(* Logix 5000 project; controller TEC_81 vendor 1 type 14 code 148 rev 36.11; software revision 36.00; part 3 of 4 *)
(* tags used below, declared in another part *)
   Abrir_Prensa_CNC_2 : BOOL;   // START CYCLE CNC 2
   AbrirInterlock_conveyor_Control : BOOL;
   AbrirInterlock_conveyor_Safety : BOOL;
   AbrirInterlock_Principal_Control : BOOL;
   AbrirInterlock_Principal_Safety : BOOL;
   Axis_1 : AXIS_CIP_DRIVE;
   Axis_2 : AXIS_CIP_DRIVE;   // Almacen 2
   Close_Griper_Fanuc : BOOL;   // Señal de Griper Cerrado Robot Fanuc
   Cmd_Axis_2 : BOOL;
   Cmd_Robot_Conv_1 : BOOL;
   Cmd_Robot_Conv_2 : BOOL;
   Cmd_YPickSafe_Alm1 : BOOL;
   Cmd_YPlaceSafe_Alm1 : BOOL;
   Cmd_YSafePos_Alm1 : BOOL;
   Cmd_YtoYOff_Alm1 : BOOL;
   Cmd_YtoYPick_Alm1 : BOOL;
   Cmd_YtoYPlace_Alm1 : BOOL;
   Cmd_YtoYPlaceOffset_Alm1 : BOOL;
   Consumeded_Signals_Conveyor_1_TEC_81 : DINT;
   Conveyor_1_Tomar_Pieza : BOOL;   // Señal del Conveyor 1 para Tomar Pieza Iniciar Ciclo
   Conveyor_2_Tomar_Pieza : BOOL;   // Señal del Conveyor 2 para Tomar Pieza Iniciar Ciclo
   Destino_Fanuc_Wait : BOOL;
   EStops_OK : BOOL;
   EStops_OK_External : DINT;
   Fanuc_Confirma_Dejar_Pieza : BOOL;   // Confirmación del Robot Fanuc para dejar la pieza
   Fanuc_Confirma_Retraido : BOOL;   // Señal de Fanuc en posición segura en Mesa Kuka
   Fanuc_Confirma_Tomar_Pieza : BOOL;   // Señal de Fanuc en posición para Tomar pieza
   From_Robot : FromRobot_v02;
   From_Wh2 : DINT;
   FromStorage1 : DINT;
   Home_Sensor : BOOL;
   Input_Reset_Almacen_1 : BOOL;
   Input_Reset_almacen_2 : BOOL;
   Input_Reset_Principal : BOOL;
   Input_Reset_Salida_1 : BOOL;
   Int_Robot_2 : INT;
   Interlocks_Ok : BOOL;
   LigthCurtain_ok : BOOL;
   MC_1_EStop : DCI_STOP;
   MC_1_EStop_Status : BOOL;
   MC_1_Interlock : DCI_STOP;
   MC_1_Interlock_Status : BOOL;
   MC_1_LigthCurtain : DCI_STOP;
   MC_1_LigthCurtain_Status : BOOL;
   MC_2_EStop : DCI_STOP;
   MC_2_EStop_Status : BOOL;
   MC_2_Interlock : DCI_STOP;
   MC_2_Interlock_Status : BOOL;
   MC_2_LightCurtain_Status : BOOL;
   MC_2_LigthCurtain : DCI_STOP;
   MC_3_EStop : DCI_STOP;
   MC_3_EStop_Status : BOOL;
   MC_4_EStop : DCI_STOP;
   MC_4_EStop_Status : BOOL;
   MC_5_EStop : DCI_STOP;
   MC_5_EStop_Status : BOOL;
   ok : BOOL;
   Open_Griper_Fanuc : BOOL;   // Señal De Griper Abierto Robot Fanuc
   Produced_Signals_TEC_81_Conveyor_1 : DINT;
   Puerta_Abierta_CNC_1 : BOOL;   // Sensor de Puerta Abierta en CNC 1 Conveyor 1
   Puerta_Abierta_CNC_2 : BOOL;   // Sensor de Puerta Abierta en CNC 2 Conveyor 2
   Reset_Almacen_1 : BOOL;
   Reset_almacen_2 : BOOL;
   Reset_Principal : BOOL;
   Reset_Salida_1 : BOOL;
   Retorno_Pieza_A_Conveyor_1 : BOOL;
   Robot_Step : DINT;
   Safety_FromTEC81 : Safety;
   SafetyReset_almacen_1 : BOOL;
   SafetyReset_almacen_2 : BOOL;
   SafetyReset_Principal : BOOL;
   SafetyReset_Salida_1 : BOOL;
   Sensor_Griper_Fanuc_Abierto : BOOL;   // Sensor Indicador Griper en Robot Fanuc Abierto
   Sensor_Griper_Fanuc_Cerrado : BOOL;   // Sensor Indicador Griper en Robot Fanuc Cerrado
   Sensor_Piston_2_Ext_Mesa : BOOL;   // Sensor de Pistón Extendido Centro de la Mesa Central
   Sensor_Piston_2_Ret_Mesa : BOOL;   // Sensor de Pistón Retraido Centro de la Mesa Central
   Signal_Fanuc_Tomar_Pieza_Conv_1 : BOOL;   // Señal para Tomar pieza desde el Conveyor 1 Hacia CNC
   Storage_1_Y_ActualPosition : REAL;
   Storage_2_Y_ActualPosition : REAL;
   Tec81_to_Wh2 : DINT;
   test_com : BOOL;   // bit e comunicacion
   TEst_Leaa_Sfty : DINT;
   To_Robot : ToRobot;
   TT : BOOL;

PROGRAM MainProgram   (* main routine MainRoutine *)

ROUTINE _01_Inputs   (* ladder *)
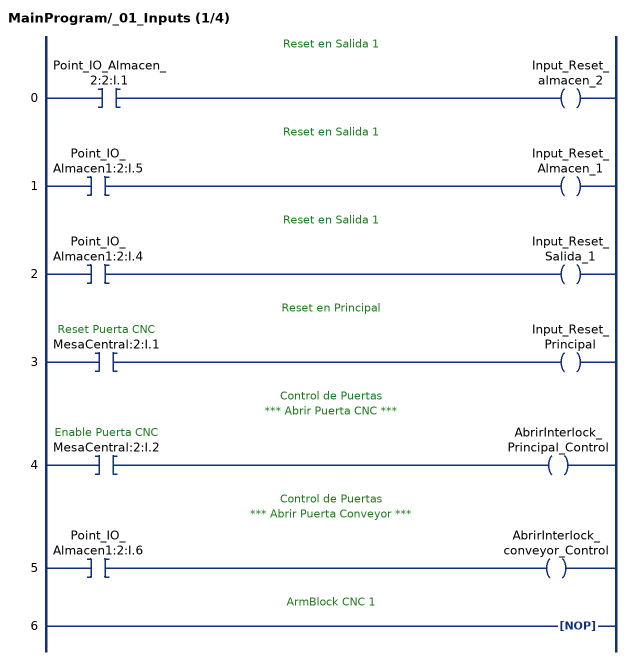
   // Reset en Salida 1
   0: XIC(Point_IO_Almacen_2:2:I.1)OTE(Input_Reset_almacen_2);
   // Reset en Salida 1
   1: XIC(Point_IO_Almacen1:2:I.5)OTE(Input_Reset_Almacen_1);
   // Reset en Salida 1
   2: XIC(Point_IO_Almacen1:2:I.4)OTE(Input_Reset_Salida_1);
   // Reset en Principal
   3: XIC(MesaCentral:2:I.1)OTE(Input_Reset_Principal);
   // Control de Puertas
   // *** Abrir Puerta CNC ***
   4: XIC(MesaCentral:2:I.2)OTE(AbrirInterlock_Principal_Control);
   // Control de Puertas
   // *** Abrir Puerta Conveyor ***
   5: XIC(Point_IO_Almacen1:2:I.6)OTE(AbrirInterlock_conveyor_Control);
   // ArmBlock CNC 1
   6: NOP();
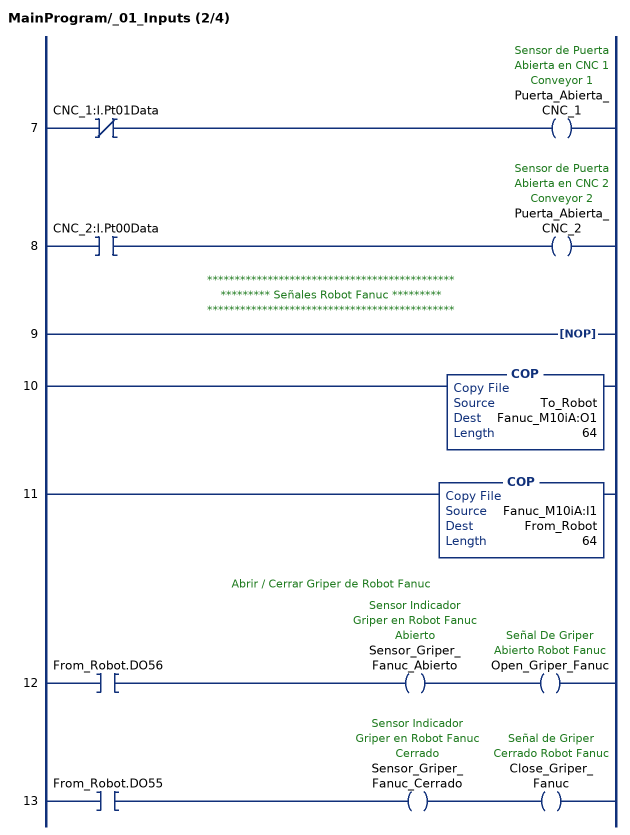
   7: XIO(CNC_1:I.Pt01Data)OTE(Puerta_Abierta_CNC_1);
   8: XIC(CNC_2:I.Pt00Data)OTE(Puerta_Abierta_CNC_2);
   // *********************************************
   // ********* Señales Robot Fanuc *********
   // *********************************************
   9: NOP();
   10: COP(To_Robot,Fanuc_M10iA:O1,64);
   11: COP(Fanuc_M10iA:I1,From_Robot,64);
   // Abrir / Cerrar Griper de Robot Fanuc
   12: XIC(From_Robot.DO56)OTE(Sensor_Griper_Fanuc_Abierto)OTE(Open_Griper_Fanuc);
   13: XIC(From_Robot.DO55)OTE(Sensor_Griper_Fanuc_Cerrado)OTE(Close_Griper_Fanuc);
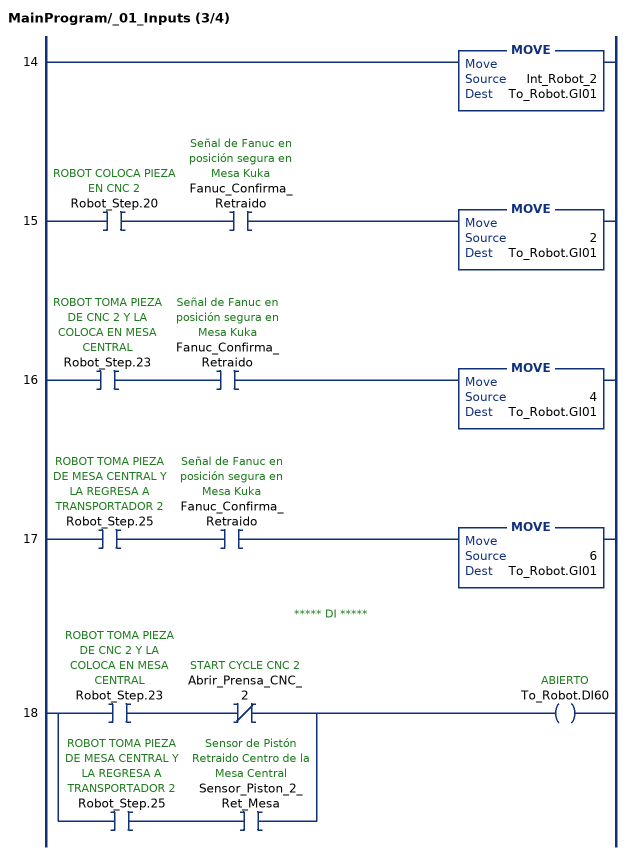
   14: MOVE(Int_Robot_2,To_Robot.GI01);
   15: XIC(Robot_Step.20)XIC(Fanuc_Confirma_Retraido)MOVE(2,To_Robot.GI01);
   16: XIC(Robot_Step.23)XIC(Fanuc_Confirma_Retraido)MOVE(4,To_Robot.GI01);
   17: XIC(Robot_Step.25)XIC(Fanuc_Confirma_Retraido)MOVE(6,To_Robot.GI01);
   // ***** DI *****
   18: [XIC(Robot_Step.23) XIO(Abrir_Prensa_CNC_2) ,XIC(Robot_Step.25) XIC(Sensor_Piston_2_Ret_Mesa) ]OTE(To_Robot.DI60);
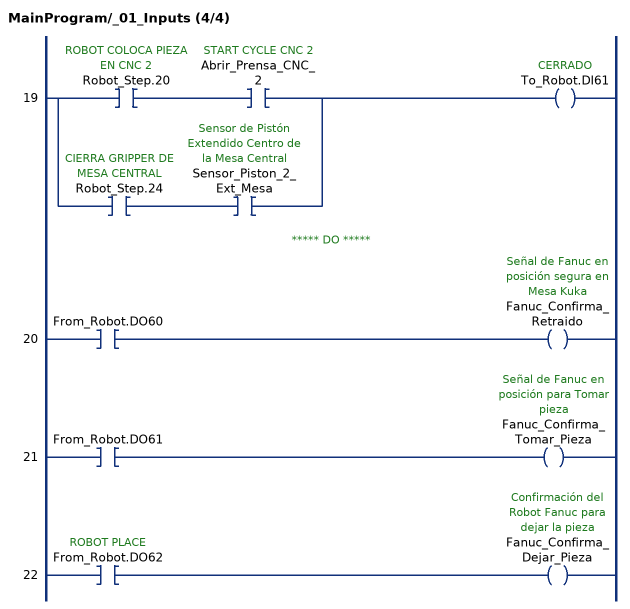
   19: [XIC(Robot_Step.20) XIC(Abrir_Prensa_CNC_2) ,XIC(Robot_Step.24) XIC(Sensor_Piston_2_Ext_Mesa) ]OTE(To_Robot.DI61);
   // ***** DO *****
   20: XIC(From_Robot.DO60)OTE(Fanuc_Confirma_Retraido);
   21: XIC(From_Robot.DO61)OTE(Fanuc_Confirma_Tomar_Pieza);
   22: XIC(From_Robot.DO62)OTE(Fanuc_Confirma_Dejar_Pieza);
END_ROUTINE

ROUTINE _06_Fanuc_States   (* ladder *)
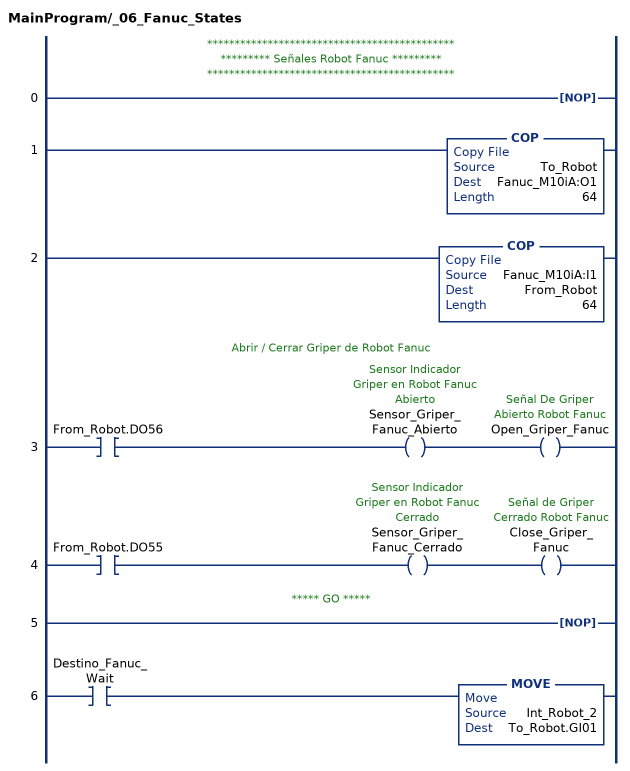
   // *********************************************
   // ********* Señales Robot Fanuc *********
   // *********************************************
   0: NOP();
   1: COP(To_Robot,Fanuc_M10iA:O1,64);
   2: COP(Fanuc_M10iA:I1,From_Robot,64);
   // Abrir / Cerrar Griper de Robot Fanuc
   3: XIC(From_Robot.DO56)OTE(Sensor_Griper_Fanuc_Abierto)OTE(Open_Griper_Fanuc);
   4: XIC(From_Robot.DO55)OTE(Sensor_Griper_Fanuc_Cerrado)OTE(Close_Griper_Fanuc);
   // ***** GO *****
   5: NOP();
   6: XIC(Destino_Fanuc_Wait)MOVE(Int_Robot_2,To_Robot.GI01);
END_ROUTINE

ROUTINE _08_Outputs   (* ladder *)
END_ROUTINE

ROUTINE _09_Resets   (* ladder *)
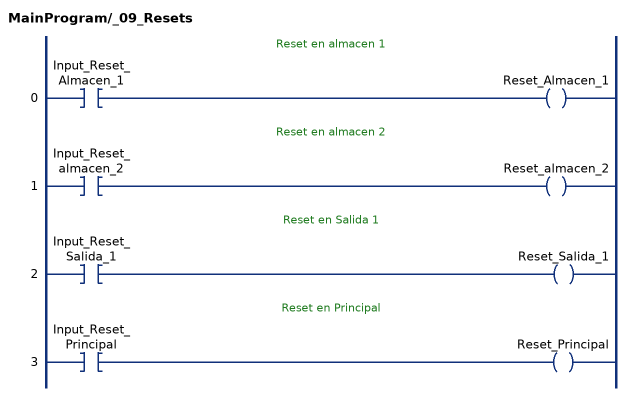
   // Reset en almacen 1
   0: XIC(Input_Reset_Almacen_1)OTE(Reset_Almacen_1);
   // Reset en almacen 2
   1: XIC(Input_Reset_almacen_2)OTE(Reset_almacen_2);
   // Reset en Salida 1
   2: XIC(Input_Reset_Salida_1)OTE(Reset_Salida_1);
   // Reset en Principal
   3: XIC(Input_Reset_Principal)OTE(Reset_Principal);
END_ROUTINE

ROUTINE _10_ExternalComm   (* ladder *)
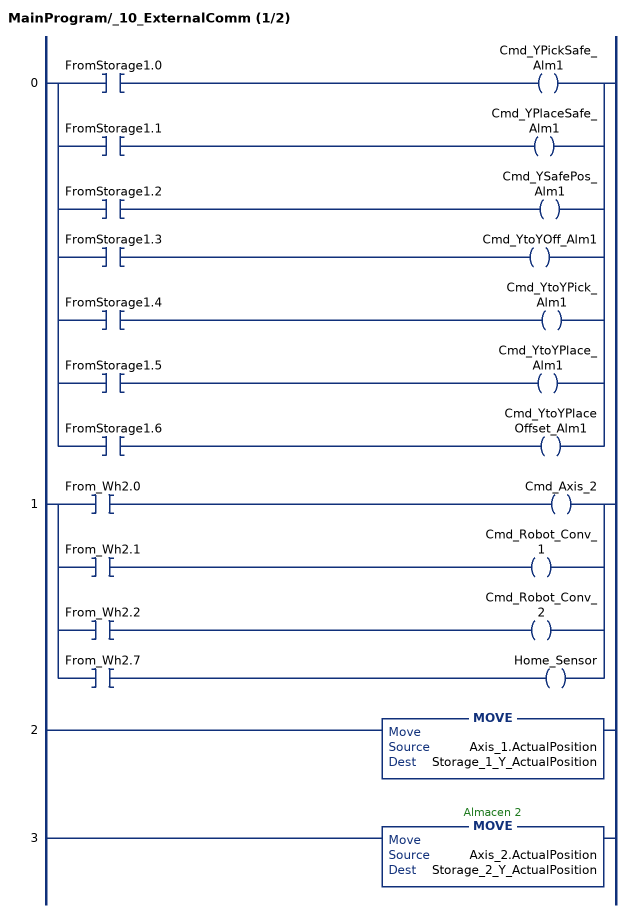
   0: [XIC(FromStorage1.0) OTE(Cmd_YPickSafe_Alm1) ,XIC(FromStorage1.1) OTE(Cmd_YPlaceSafe_Alm1) ,XIC(FromStorage1.2) OTE(Cmd_YSafePos_Alm1) ,XIC(FromStorage1.3) OTE(Cmd_YtoYOff_Alm1) ,XIC(FromStorage1.4) OTE(Cmd_YtoYPick_Alm1) ,XIC(FromStorage1.5) OTE(Cmd_YtoYPlace_Alm1) ,XIC(FromStorage1.6) OTE(Cmd_YtoYPlaceOffset_Alm1) ];
   1: [XIC(From_Wh2.0) OTE(Cmd_Axis_2) ,XIC(From_Wh2.1) OTE(Cmd_Robot_Conv_1) ,XIC(From_Wh2.2) OTE(Cmd_Robot_Conv_2) ,XIC(From_Wh2.7) OTE(Home_Sensor) ];
   2: MOVE(Axis_1.ActualPosition,Storage_1_Y_ActualPosition);
   3: MOVE(Axis_2.ActualPosition,Storage_2_Y_ActualPosition);
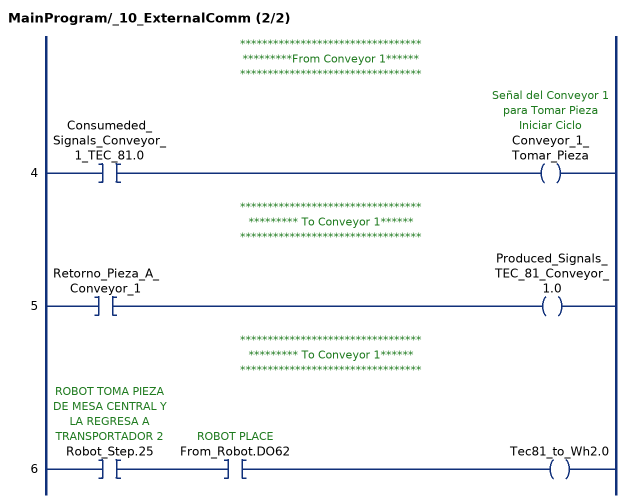
   // *********************************
   // *********From Conveyor 1******
   // *********************************
   4: XIC(Consumeded_Signals_Conveyor_1_TEC_81.0)OTE(Conveyor_1_Tomar_Pieza);
   // *********************************
   // ********* To Conveyor 1******
   // *********************************
   5: XIC(Retorno_Pieza_A_Conveyor_1)OTE(Produced_Signals_TEC_81_Conveyor_1.0);
   // *********************************
   // ********* To Conveyor 1******
   // *********************************
   6: XIC(Robot_Step.25)XIC(From_Robot.DO62)OTE(Tec81_to_Wh2.0);
END_ROUTINE

ROUTINE _11_External   (* ladder *)
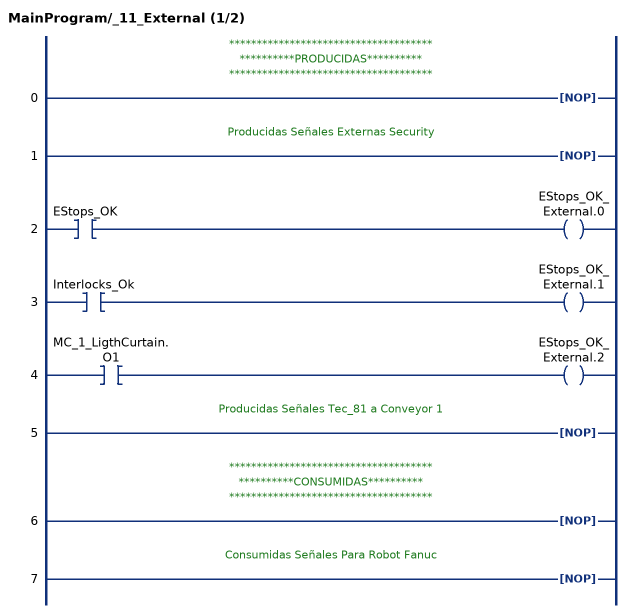
   // *************************************
   // **********PRODUCIDAS**********
   // *************************************
   0: NOP();
   // Producidas Señales Externas Security
   1: NOP();
   2: XIC(EStops_OK)OTE(EStops_OK_External.0);
   3: XIC(Interlocks_Ok)OTE(EStops_OK_External.1);
   4: XIC(MC_1_LigthCurtain.O1)OTE(EStops_OK_External.2);
   // Producidas Señales Tec_81 a Conveyor 1
   5: NOP();
   // *************************************
   // **********CONSUMIDAS**********
   // *************************************
   6: NOP();
   // Consumidas Señales Para Robot Fanuc
   7: NOP();
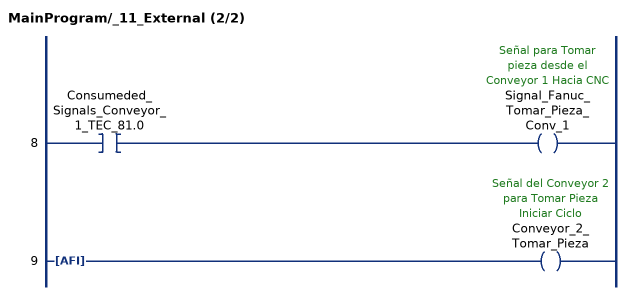
   8: XIC(Consumeded_Signals_Conveyor_1_TEC_81.0)OTE(Signal_Fanuc_Tomar_Pieza_Conv_1);
   9: AFI()OTE(Conveyor_2_Tomar_Pieza);
END_ROUTINE

ROUTINE MainRoutine   (* ladder *)
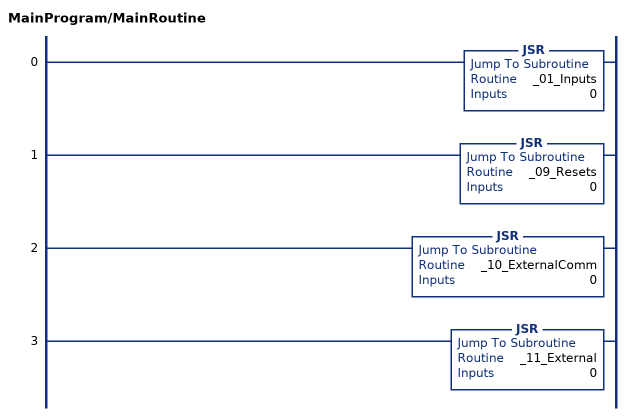
   0: JSR(_01_Inputs,0);
   1: JSR(_09_Resets,0);
   2: JSR(_10_ExternalComm,0);
   3: JSR(_11_External,0);
END_ROUTINE
END_PROGRAM

PROGRAM SafetyProgram   (* main routine MainRoutine, safety *)
VAR
   dummy : BOOL;
   Safety_Close_Loop_ok : BOOL := 1;
   Safety_Latch_Timer : TIMER := (PRE := 500);
   Safety_Reset_General : BOOL;
   test_1 : BOOL;
   test_21 : BOOL;
   TOF_STO_KinetixStorage1 : TIMER := (PRE := 10000, EN := 1, DN := 1);
END_VAR

ROUTINE Estops   (* ladder *)
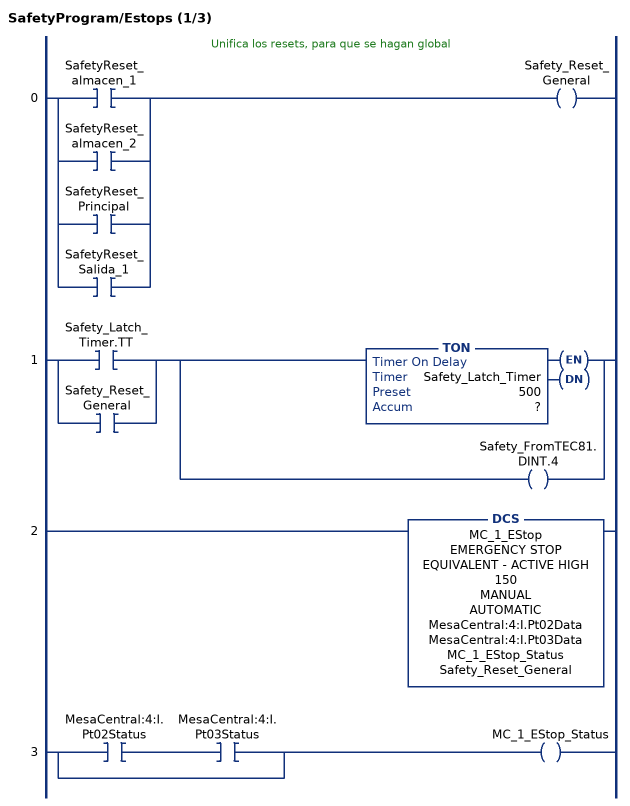
   // Unifica los resets, para que se hagan global
   0: [XIC(SafetyReset_almacen_1) ,XIC(SafetyReset_almacen_2) ,XIC(SafetyReset_Principal) ,XIC(SafetyReset_Salida_1) ]OTE(Safety_Reset_General);
   1: [XIC(Safety_Latch_Timer.TT) ,XIC(Safety_Reset_General) ][TON(Safety_Latch_Timer,?,?) ,OTE(Safety_FromTEC81.DINT.4) ];
   2: DCS(MC_1_EStop,EMERGENCY STOP,EQUIVALENT - ACTIVE HIGH,150,MANUAL,AUTOMATIC,MesaCentral:4:I.Pt02Data,MesaCentral:4:I.Pt03Data,MC_1_EStop_Status,Safety_Reset_General);
   3: [XIC(MesaCentral:4:I.Pt02Status) XIC(MesaCentral:4:I.Pt03Status) ,]OTE(MC_1_EStop_Status);
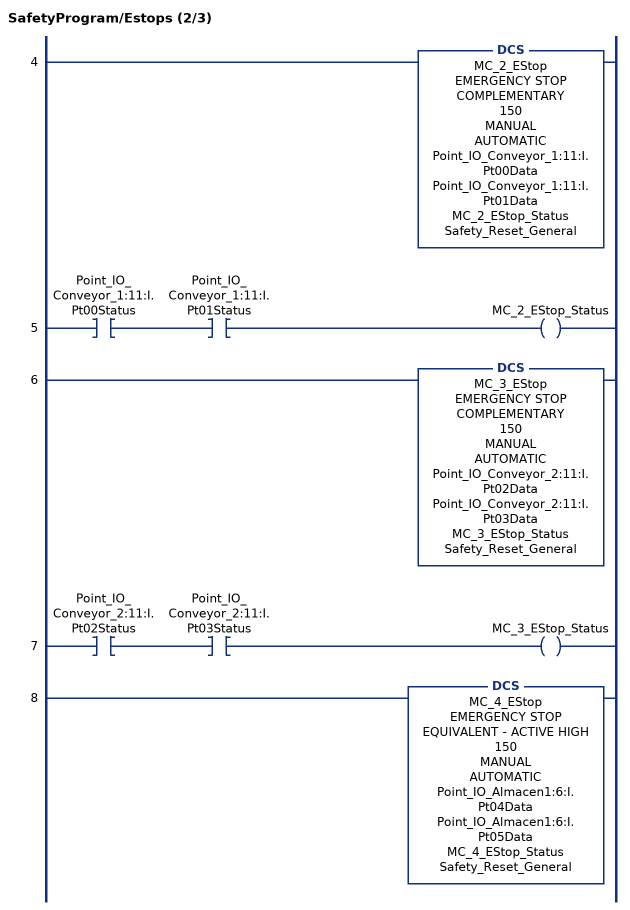
   4: DCS(MC_2_EStop,EMERGENCY STOP,COMPLEMENTARY,150,MANUAL,AUTOMATIC,Point_IO_Conveyor_1:11:I.Pt00Data,Point_IO_Conveyor_1:11:I.Pt01Data,MC_2_EStop_Status,Safety_Reset_General);
   5: XIC(Point_IO_Conveyor_1:11:I.Pt00Status)XIC(Point_IO_Conveyor_1:11:I.Pt01Status)OTE(MC_2_EStop_Status);
   6: DCS(MC_3_EStop,EMERGENCY STOP,COMPLEMENTARY,150,MANUAL,AUTOMATIC,Point_IO_Conveyor_2:11:I.Pt02Data,Point_IO_Conveyor_2:11:I.Pt03Data,MC_3_EStop_Status,Safety_Reset_General);
   7: XIC(Point_IO_Conveyor_2:11:I.Pt02Status)XIC(Point_IO_Conveyor_2:11:I.Pt03Status)OTE(MC_3_EStop_Status);
   8: DCS(MC_4_EStop,EMERGENCY STOP,EQUIVALENT - ACTIVE HIGH,150,MANUAL,AUTOMATIC,Point_IO_Almacen1:6:I.Pt04Data,Point_IO_Almacen1:6:I.Pt05Data,MC_4_EStop_Status,Safety_Reset_General);
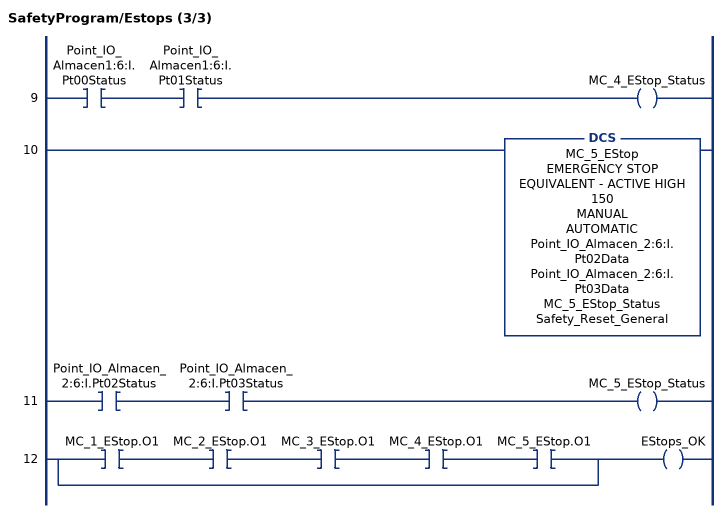
   9: XIC(Point_IO_Almacen1:6:I.Pt00Status)XIC(Point_IO_Almacen1:6:I.Pt01Status)OTE(MC_4_EStop_Status);
   10: DCS(MC_5_EStop,EMERGENCY STOP,EQUIVALENT - ACTIVE HIGH,150,MANUAL,AUTOMATIC,Point_IO_Almacen_2:6:I.Pt02Data,Point_IO_Almacen_2:6:I.Pt03Data,MC_5_EStop_Status,Safety_Reset_General);
   11: XIC(Point_IO_Almacen_2:6:I.Pt02Status)XIC(Point_IO_Almacen_2:6:I.Pt03Status)OTE(MC_5_EStop_Status);
   12: [XIC(MC_1_EStop.O1) XIC(MC_2_EStop.O1) XIC(MC_3_EStop.O1) XIC(MC_4_EStop.O1) XIC(MC_5_EStop.O1) ,]OTE(EStops_OK);
END_ROUTINE

ROUTINE External_COMM   (* ladder *)
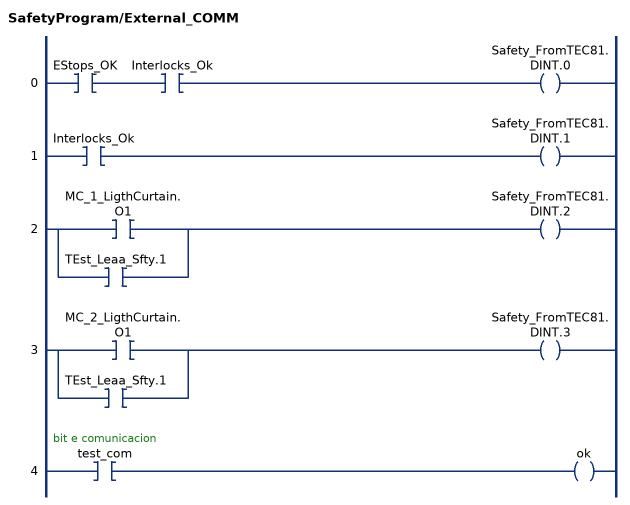
   0: XIC(EStops_OK)XIC(Interlocks_Ok)OTE(Safety_FromTEC81.DINT.0);
   1: XIC(Interlocks_Ok)OTE(Safety_FromTEC81.DINT.1);
   2: [XIC(MC_1_LigthCurtain.O1) ,XIC(TEst_Leaa_Sfty.1) ]OTE(Safety_FromTEC81.DINT.2);
   3: [XIC(MC_2_LigthCurtain.O1) ,XIC(TEst_Leaa_Sfty.1) ]OTE(Safety_FromTEC81.DINT.3);
   4: XIC(test_com)OTE(ok);
END_ROUTINE

ROUTINE Interlocks   (* ladder *)
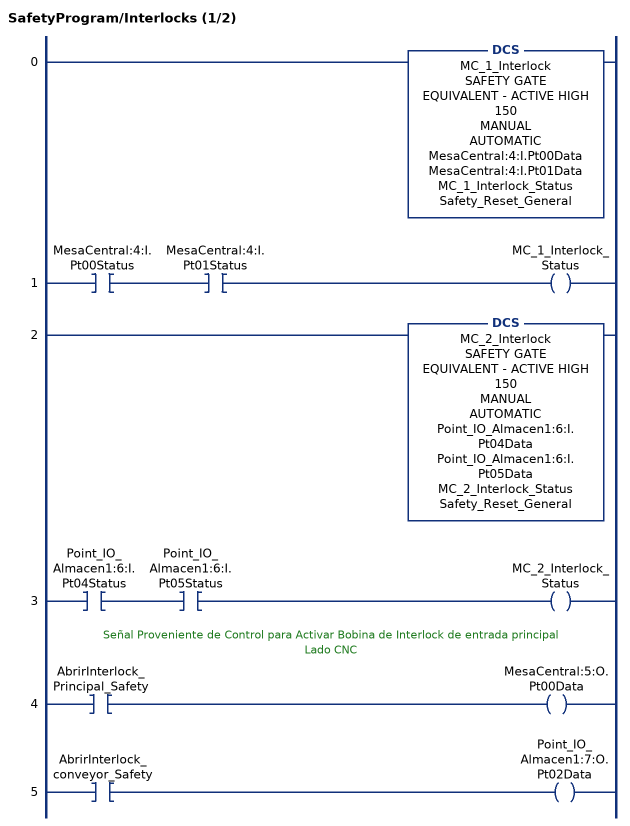
   0: DCS(MC_1_Interlock,SAFETY GATE,EQUIVALENT - ACTIVE HIGH,150,MANUAL,AUTOMATIC,MesaCentral:4:I.Pt00Data,MesaCentral:4:I.Pt01Data,MC_1_Interlock_Status,Safety_Reset_General);
   1: XIC(MesaCentral:4:I.Pt00Status)XIC(MesaCentral:4:I.Pt01Status)OTE(MC_1_Interlock_Status);
   2: DCS(MC_2_Interlock,SAFETY GATE,EQUIVALENT - ACTIVE HIGH,150,MANUAL,AUTOMATIC,Point_IO_Almacen1:6:I.Pt04Data,Point_IO_Almacen1:6:I.Pt05Data,MC_2_Interlock_Status,Safety_Reset_General);
   3: XIC(Point_IO_Almacen1:6:I.Pt04Status)XIC(Point_IO_Almacen1:6:I.Pt05Status)OTE(MC_2_Interlock_Status);
   // Señal Proveniente de Control para Activar Bobina de Interlock de entrada principal
   // Lado CNC
   4: XIC(AbrirInterlock_Principal_Safety)OTE(MesaCentral:5:O.Pt00Data);
   5: XIC(AbrirInterlock_conveyor_Safety)OTE(Point_IO_Almacen1:7:O.Pt02Data);
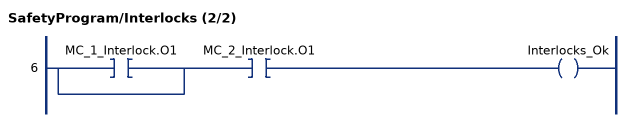
   6: [XIC(MC_1_Interlock.O1) ,]XIC(MC_2_Interlock.O1)OTE(Interlocks_Ok);
END_ROUTINE

ROUTINE LigthCurrtains   (* ladder *)
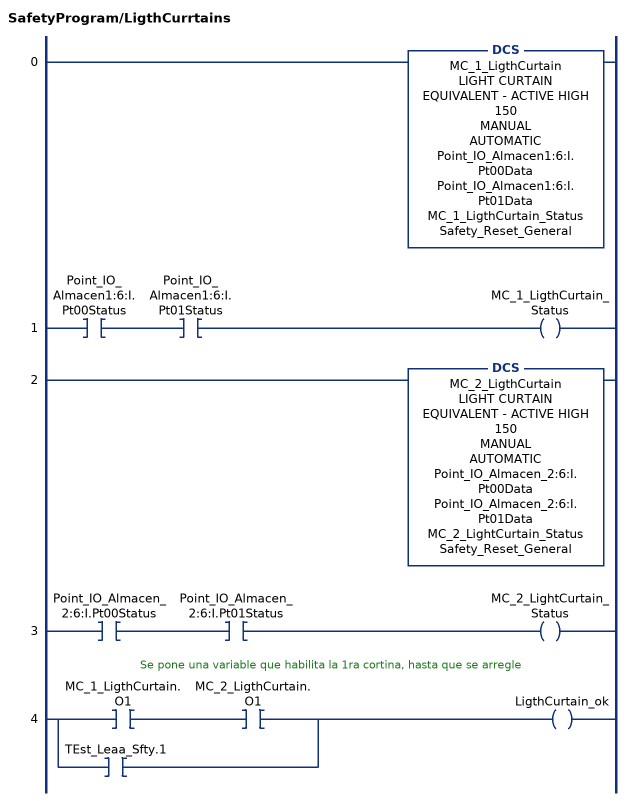
   0: DCS(MC_1_LigthCurtain,LIGHT CURTAIN,EQUIVALENT - ACTIVE HIGH,150,MANUAL,AUTOMATIC,Point_IO_Almacen1:6:I.Pt00Data,Point_IO_Almacen1:6:I.Pt01Data,MC_1_LigthCurtain_Status,Safety_Reset_General);
   1: XIC(Point_IO_Almacen1:6:I.Pt00Status)XIC(Point_IO_Almacen1:6:I.Pt01Status)OTE(MC_1_LigthCurtain_Status);
   2: DCS(MC_2_LigthCurtain,LIGHT CURTAIN,EQUIVALENT - ACTIVE HIGH,150,MANUAL,AUTOMATIC,Point_IO_Almacen_2:6:I.Pt00Data,Point_IO_Almacen_2:6:I.Pt01Data,MC_2_LightCurtain_Status,Safety_Reset_General);
   3: XIC(Point_IO_Almacen_2:6:I.Pt00Status)XIC(Point_IO_Almacen_2:6:I.Pt01Status)OTE(MC_2_LightCurtain_Status);
   // Se pone una variable que habilita la 1ra cortina, hasta que se arregle
   4: [XIC(MC_1_LigthCurtain.O1) XIC(MC_2_LigthCurtain.O1) ,XIC(TEst_Leaa_Sfty.1) ]OTE(LigthCurtain_ok);
END_ROUTINE
